PROGRAM prgComEffIO
VAR
	fbCom		: FB_MqttCommunicator_V2;
END_VAR

fbCom(
	bConnect:= TRUE, 
	strAuthKey := 'BE736352867778',
	sUserName:= '9e35a788-9544-4d1e-a992-8e2eed9a2bf4', 
	sUserPassword:= 'b22fd0d3-05b2-481b-ab97-9bb6cc09e5f2', 
	eSavePositionCertificate:= eSavePositionOnPLC.ePostionHardDisk, 
	bConnected=> , 
	bError=> , 
	hrErrorCode=> , 
	eConnectionState=> , 
	eErrorMessage_Out=> );

END_PROGRAM

(* stored: Version 1.1.0.1, ProductVersion 3.1.4024.11
   POU prgComEffIO: Id {cbcd318b-bf51-484c-bcaa-d6efcdf43fe3}, SpecialFunc None *)
